// TIA Portal V17 export
// export: Created 2025-03-10T13:12:01.3367506Z, ExportSetting WithDefaults, DisplayName Totally Integrated Automation Portal, DisplayVersion V17 Update 8, DisplayName TIA Portal Openness, DisplayVersion V17 Update 8, DisplayName TIA Portal Version Control Interface, DisplayVersion V17, DisplayName SINAMICS Startdrive Advanced, DisplayVersion V17 SP2, DisplayName SINAMICS Startdrive G110M, G120, G120C, G120D, G120P, G115D, DisplayVersion V17 SP2, DisplayName SINAMICS Startdrive G130, G150, S120, S150, SINAMICS MV, S210, DisplayVersion V17 SP2, DisplayName STEP 7 Professional, DisplayVersion V17 Update 8, DisplayName SINUMERIK ONE STEP 7 Toolbox, DisplayVersion V17 Update 12, DisplayName SINUMERIK 840D sl STEP 7 Toolbox, DisplayVersion V17 Update 12, DisplayName STEP 7 Safety, DisplayVersion V17 Update 6, DisplayName WinCC Advanced, DisplayVersion V17 Update 8
TYPE "LBP_typePowerrideConfig"
TITLE = Data type for configuration of Powerride / Tipo de datos para configuración de Powerride / Datentyp für Konfiguration von Powerride
// User data type for LBP_PowerrideConfig / Tipo de datos de usuario para LBP_PowerrideConfig / Anwenderdatentyp für LBP_PowerrideConfig
// stored: IsFailsafeCompliant false
   STRUCT
      pos100 { S7_SetPoint := 'True'} : USInt := 0;   // [1...36] Schalterposition bei 100 % Override / [1..36] switch position at 100% ovr / [1...36] Posición de interruptor en 100 % de corrección
      posMax { S7_SetPoint := 'True'} : USInt := 0;   // [1...36] Schalterposition bei max. Override / [1..36] switch position at maximum ovr / [1...36] Posición de interruptor en corrección máx.
      delay100 { S7_SetPoint := 'True'} : Time := T#500MS;   // Verzögerung bei 100 % vor Fortsetzen des Override / time delay at 100% before continuing ovr / Retardo en 100 % antes de continuar la corrección
      switchPos { S7_SetPoint := 'True'} : Array[1..36] of "LBP_typePowerrideConfigPos";   // Wert, Farbe und Vibration für Position / value, colour and vibration for position / Valor, color y vibración para posición
   END_STRUCT;
END_TYPE
